FUNCTION_BLOCK AX_E_SWITCH (* Switching (demultiplexing) an event based on boolean input G *)
  (* Standard: 61499-2; Description: Copyright (c) 2025 HR Agrartechnik GmbH This program and the accompanying materials are made available under the terms of the Eclipse Public License 2.0 which is available at https://www.eclipse.org/legal/epl-2.0/ SPDX-License-Identifier: EPL-2.0 *)
  (* Version 1.0, 2025-01-24, Franz Höpfinger, HR Agrartechnik GmbH *)
  PACKAGE adapter::events::unidirectional;
  IMPORT eclipse4diac::core::TypeHash;
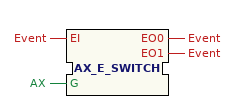
  EVENT_INPUT
    EI; (* Event Input *)
  END_EVENT
  EVENT_OUTPUT
    EO0; (* Output, switched from EI when G=0 *)
    EO1; (* Output, switched from EI when G=1 *)
  END_EVENT
  SOCKETS
    G : adapter::types::unidirectional::AX; (* Switch EI to EI0 when G=0, to EI1 when G=1 *)
  END_SOCKETS
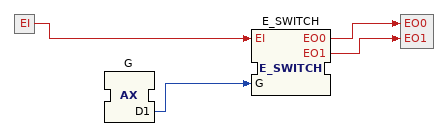
  FBS
    E_SWITCH : iec61499::events::E_SWITCH;
  END_FBS
  EVENT_CONNECTIONS
    EI TO E_SWITCH.EI;
    E_SWITCH.EO0 TO EO0;
    E_SWITCH.EO1 TO EO1;
  END_CONNECTIONS
  DATA_CONNECTIONS
    G.D1 TO E_SWITCH.G;
  END_CONNECTIONS
END_FUNCTION_BLOCK
